PROGRAM set_pos
VAR
	MC_SetPosition1: MC_SetPosition;
	MC_SetPosition2: MC_SetPosition;
	MC_SetPosition3: MC_SetPosition;
	MC_SetPosition4: MC_SetPosition;
	MC_SetPosition5: MC_SetPosition;
	MC_SetPosition6: MC_SetPosition;
END_VAR

MC_SetPosition1(
	Axis:= axis.Axis1, 
	Execute:= , 
	Position:= , 
	Mode:= , 
	Options:= , 
	Done=> , 
	Busy=> , 
	Error=> , 
	ErrorID=> );

MC_SetPosition2(
	Axis:= axis.Axis2, 
	Execute:= , 
	Position:= , 
	Mode:= , 
	Options:= , 
	Done=> , 
	Busy=> , 
	Error=> , 
	ErrorID=> );
	
MC_SetPosition3(
	Axis:= axis.Axis3, 
	Execute:= , 
	Position:= , 
	Mode:= , 
	Options:= , 
	Done=> , 
	Busy=> , 
	Error=> , 
	ErrorID=> );

MC_SetPosition4(
	Axis:= axis.Axis4, 
	Execute:= , 
	Position:= , 
	Mode:= , 
	Options:= , 
	Done=> , 
	Busy=> , 
	Error=> , 
	ErrorID=> );
	
MC_SetPosition5(
	Axis:= axis.Axis5, 
	Execute:= , 
	Position:= , 
	Mode:= , 
	Options:= , 
	Done=> , 
	Busy=> , 
	Error=> , 
	ErrorID=> );

MC_SetPosition6(
	Axis:= axis.Axis6, 
	Execute:= , 
	Position:= , 
	Mode:= , 
	Options:= , 
	Done=> , 
	Busy=> , 
	Error=> , 
	ErrorID=> );

END_PROGRAM

(* stored: Version 1.1.0.1, ProductVersion 3.1.4024.0
   POU set_pos: Id {97549c07-bd89-41b0-baec-8d1d12a907c4}, SpecialFunc None *)
